(* Logix 5000 project; controller ARS14002_PLC vendor 1 type 14 code 218 rev 30.11; software revision 30.01; part 5 of 13 *)
(* tags used below, declared in another part *)
   AN_1000C : CM_AI_SCL;
   AN_1000C_RESTART_TMR : TIMER;
   AN_1000C_SP : INT;
   AN_1000C_STOP_TMR : TIMER;
   AN_101_PERMISSIVE_AUTO : BOOL;   // Does the PLC look at AN-101
   AN_101A : CM_AI_SCL;
   AN_101A_RESTART_TIME : REAL;
   AN_101A_RESTART_TMR : TIMER;
   AN_101A_SP : REAL;
   AN_101A_STOP_TIME : REAL;
   AN_101A_STOP_TMR : TIMER;
   AN_101B : CM_AI_SCL;
   AN_101B_RESTART_TIME : REAL;
   AN_101B_RESTART_TMR : TIMER;
   AN_101B_SP : REAL;
   AN_101B_STOP_TIME : REAL;
   AN_101B_STOP_TMR : TIMER;
   AN_101C : CM_AI_SCL;
   AN_101C_RESTART_TIME : REAL;
   AN_101C_RESTART_TMR : TIMER;
   AN_101C_SP : REAL;
   AN_101C_STOP_TIME : REAL;
   AN_101C_STOP_TMR : TIMER;
   AN_200A : CM_AI_SCL;
   AN_200A_RESTART_TMR : TIMER;
   AN_200A_SP : REAL;
   AN_200A_STOP_TMR : TIMER;
   ARS_COLLECT : BOOL;
   ARS_COLLECT_AUTO : BOOL;
   ARS_DERIME_AUTO : BOOL;
   AT2_ATOMIZE_LATCH : BOOL;
   AT2_CHAMBER_PRESSURE : REAL;
   AT2_CHAMBER_PRESSURE_SP : REAL;
   AT2_PLANT_ATOMIZING : BOOL;
   AT2_PLANT_BACKFILL : BOOL;
   AT2_PLANT_COLLECT_AUTO : BOOL;
   AT2_PT_101B_Pressure_Override : REAL;   // Setpoint at which FCV_101 will open and relieve the pressure despite controls, not an interlock
   AT2_START_ATOMIZATION : BOOL;
   AT2_V1_OPEN : BOOL;
   AT2_V1_OPEN_POSTHEAT_CTR : COUNTER;
   AT2_V1_OPEN_POSTHEAT_CTR_SP : DINT;
   AT3_ATOMIZE_VALVE_OPEN : BOOL;
   AT3_CHAMBER_PRESSURE : REAL;
   AT3_CHAMBER_PRESSURE_SP : REAL;
   AT3_PLANT_ATOMIZING : BOOL;
   AT3_PLANT_BACKFILL : BOOL;
   AT3_PLANT_COLLECT_AUTO : BOOL;
   AT3_PT_101C_Press_Override : REAL;   // Pressure at which FCV101 will open despite the control scheme, not an interlock
   AT3_V1_OPEN : BOOL;
   Collect_Stop_AT2_O2 : BOOL;
   Collect_Stop_AT3_O2 : BOOL;
   Collect_Stop_Dew_Pt : BOOL;
   COLLECT_STOP_INIT : TIMER;
   Collect_Stop_O2 : BOOL;
   Collect_Stop_PILOT_O2 : BOOL;
   FCV_101A : CM_AO_VLV;
   FCV_101A_DLA : REAL;
   FCV_101A_DLA_BUMP_TMR : TIMER;
   FCV_101A_DLA_TMR : TIMER;
   FCV_101A_STARTPOS : REAL;
   FCV_101B : CM_AO_VLV;
   FCV_101B_DLA : REAL;
   FCV_101B_DLA_BUMP_TMR : TIMER;
   FCV_101B_DLA_TMR : TIMER;
   FCV_101B_STARTPOS : REAL;
   FCV_101C : CM_AO_VLV;
   FCV_101C_DLA : REAL;
   FCV_101C_DLA_BUMP_TMR : TIMER;
   FCV_101C_DLA_TMR : TIMER;
   FCV_101C_STARTPOS : REAL;
   FCV_102A : CM_AO_VLV;
   FCV_102A_AT_STARTPOS : BOOL;
   FCV_102A_SP_Atomize_Venting : REAL;
   FCV_102A_SP_Idle_Collecting : REAL;
   FCV_102A_STARTPOS : REAL;
   FCV_102A_STARTPOS_TIMEOUT : TIMER;
   FCV_102B : CM_AO_VLV;
   FCV_102B_AT_STARTPOS : BOOL;
   FCV_102B_SP_Atomize_Venting : REAL;
   FCV_102B_SP_Idle_Collecting : REAL;
   FCV_102B_STARTPOS : REAL;
   FCV_102B_STARTPOS_TIMEOUT : TIMER;
   FCV_102C : CM_AO_VLV;
   FCV_102C_AT_STARTPOS : BOOL;
   FCV_102C_BUMP_CLOSE_POS : REAL;
   FCV_102C_BUMPED_CLOSED : BOOL;
   FCV_102C_CLOSE_BUMP_TMR : TIMER;
   FCV_102C_SP_Atomize_Venting : REAL;
   FCV_102C_SP_Idle_Collecting : REAL;
   FCV_102C_STARTPOS : REAL;
   FCV_102C_STARTPOS_TIMEOUT : TIMER;
   FCV_204 : CM_AO_VLV;
   FCV_204_AT_STARTPOS : BOOL;
   FCV_204_ATOMIZE_INIT : TIMER;
   FCV_204_PVSWITCH : BOOL;   // 0 = PIT-201 1 = PIT-101C
   FCV_204_SP_Atomize : REAL;
   FCV_204_SP_Atomize_Venting_Only : REAL;
   FCV_204_SP_Idle : REAL;
   FCV_204_STARTPOS : REAL;
   FCV_204_STARTPOS_0 : REAL;
   FCV_STARTPOS_TIMEOUT : TIMER;
   MODE_ATOMIZE : BOOL;
   MODE_IDLE : BOOL;
   MODE_STANDBY_IDLE : BOOL;
   MODE_STANDBY_PUMPUP : BOOL;
   PIDE_101A : PID_ENHANCED;
   PIDE_101B : PID_ENHANCED;
   PIDE_101C : PID_ENHANCED;
   PIDE_102A : PID_ENHANCED;
   PIDE_102B : PID_ENHANCED;
   PIDE_102C : PID_ENHANCED;
   PIDE_204 : PID_ENHANCED;
   PILOT_ATOMIZE_VALVE_OPEN : BOOL;   // Halo Valve
   Pilot_Atomizing_Valve_Close_TON : TIMER;
   Pilot_Atomizing_Valve_Open_TON : TIMER;
   PILOT_EXHAUST_VALVE_OPEN : BOOL;
   PILOT_INLET_VALVE_OPEN : BOOL;   // Pressure Control Status (Backfill)
   Pilot_Inlet_Valve_Open_TON : TIMER;
   PILOT_PLANT_ATOMIZING : BOOL;
   PILOT_PLANT_BACKFILL : BOOL;
   PILOT_PLANT_COLLECT_AUTO : BOOL;
   PILOT_PT_101A_Pressure_Override : REAL;   // Pressure at which 101A will be allowed despite any control limitations, intended as a rescue setpoint, not an interlock
   PT_101A : CM_AI_SCL;
   PT_101B : CM_AI_SCL;
   PT_101C : CM_AI_SCL;
   PT_201 : CM_AI_SCL;
   SV_101AF : CM_DO_GENERIC;
   SV_101AN : CM_DO_GENERIC;
   SV_101AP : CM_DO_GENERIC;
   SV_101BF : CM_DO_GENERIC;
   SV_101BN : CM_DO_GENERIC;
   SV_101BP : CM_DO_GENERIC;
   SV_101CF : CM_DO_GENERIC;
   SV_101CN : CM_DO_GENERIC;
   SV_101CP : CM_DO_GENERIC;
   SV_102AF : CM_DO_GENERIC;
   SV_102BF : CM_DO_GENERIC;
   SV_102CF : CM_DO_GENERIC;
   SV_202F : CM_DO_GENERIC;
   SV_204F : CM_DO_GENERIC;
   TE_501 : CM_AI_SCL;
   TE_501_MIN_SV_202 : REAL;
   TK_700_OVERFULL_DLA_TMR : TIMER;
   XV_101B : CM_DO_VLV;
   XV_101C : CM_DO_VLV;
(* MainProgram, continued *)

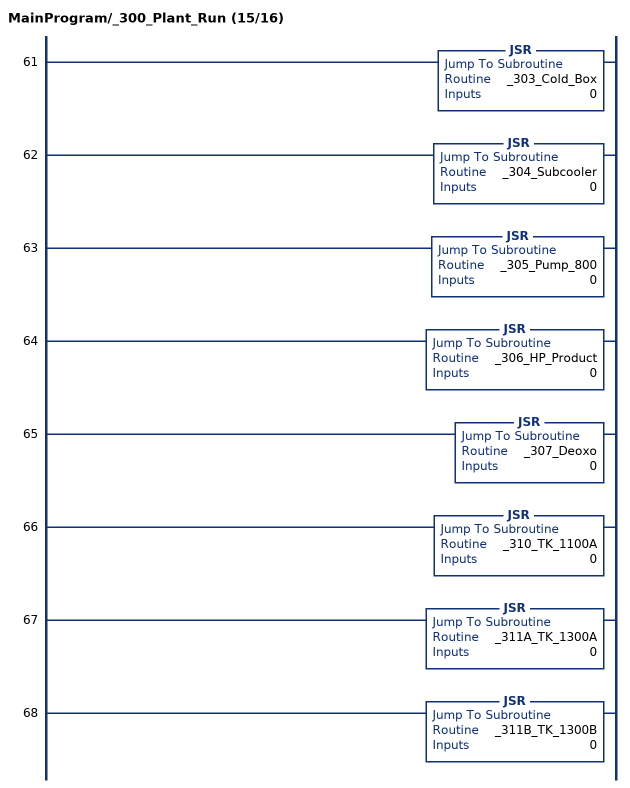
   [picture p83: MainProgram/_300_Plant_Run rungs 61-68]
   61: JSR(_303_Cold_Box,0);
   62: JSR(_304_Subcooler,0);
   63: JSR(_305_Pump_800,0);
   64: JSR(_306_HP_Product,0);
   65: JSR(_307_Deoxo,0);
   66: JSR(_310_TK_1100A,0);
   67: JSR(_311A_TK_1300A,0);
   68: JSR(_311B_TK_1300B,0);
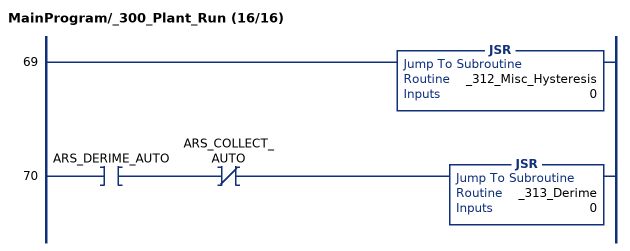
   69: JSR(_312_Misc_Hysteresis,0);
   70: XIC(ARS_DERIME_AUTO)XIO(ARS_COLLECT_AUTO)JSR(_313_Derime,0);
END_ROUTINE

ROUTINE _302_Front_End   (* ladder *)
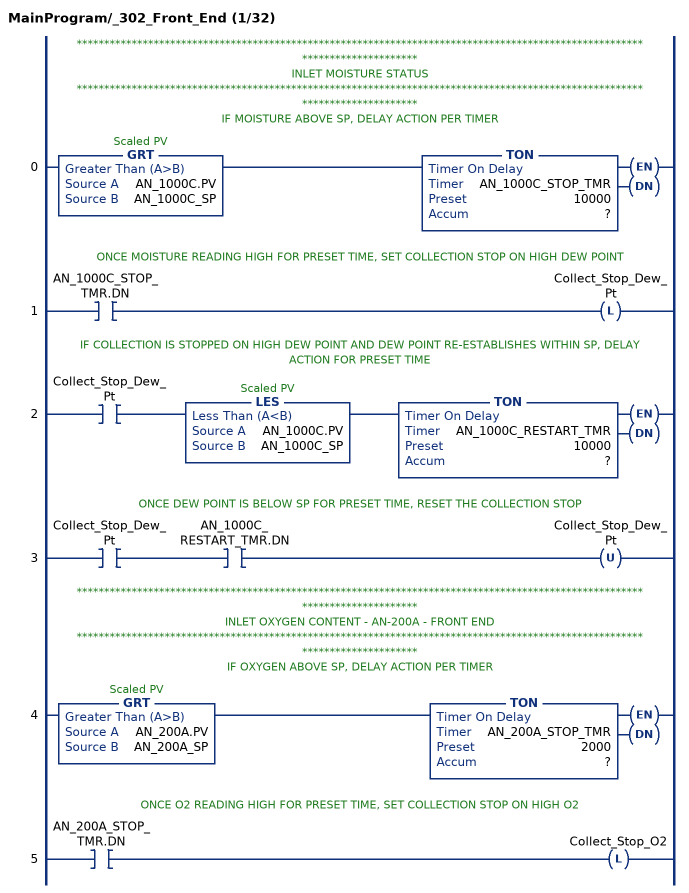
   // ****************************************************************************************************************************
   // INLET MOISTURE STATUS
   // ****************************************************************************************************************************
   // IF MOISTURE ABOVE SP, DELAY ACTION PER TIMER
   0: GRT(AN_1000C.PV,AN_1000C_SP)TON(AN_1000C_STOP_TMR,?,?);
   // ONCE MOISTURE READING HIGH FOR PRESET TIME, SET COLLECTION STOP ON HIGH DEW POINT
   1: XIC(AN_1000C_STOP_TMR.DN)OTL(Collect_Stop_Dew_Pt);
   // IF COLLECTION IS STOPPED ON HIGH DEW POINT AND DEW POINT RE-ESTABLISHES WITHIN SP, DELAY ACTION FOR PRESET TIME
   2: XIC(Collect_Stop_Dew_Pt)LES(AN_1000C.PV,AN_1000C_SP)TON(AN_1000C_RESTART_TMR,?,?);
   // ONCE DEW POINT IS BELOW SP FOR PRESET TIME, RESET THE COLLECTION STOP
   3: XIC(Collect_Stop_Dew_Pt)XIC(AN_1000C_RESTART_TMR.DN)OTU(Collect_Stop_Dew_Pt);
   // ****************************************************************************************************************************
   // INLET OXYGEN CONTENT - AN-200A - FRONT END
   // ****************************************************************************************************************************
   // IF OXYGEN ABOVE SP, DELAY ACTION PER TIMER
   4: GRT(AN_200A.PV,AN_200A_SP)TON(AN_200A_STOP_TMR,?,?);
   // ONCE O2 READING HIGH FOR PRESET TIME, SET COLLECTION STOP ON HIGH O2
   5: XIC(AN_200A_STOP_TMR.DN)OTL(Collect_Stop_O2);
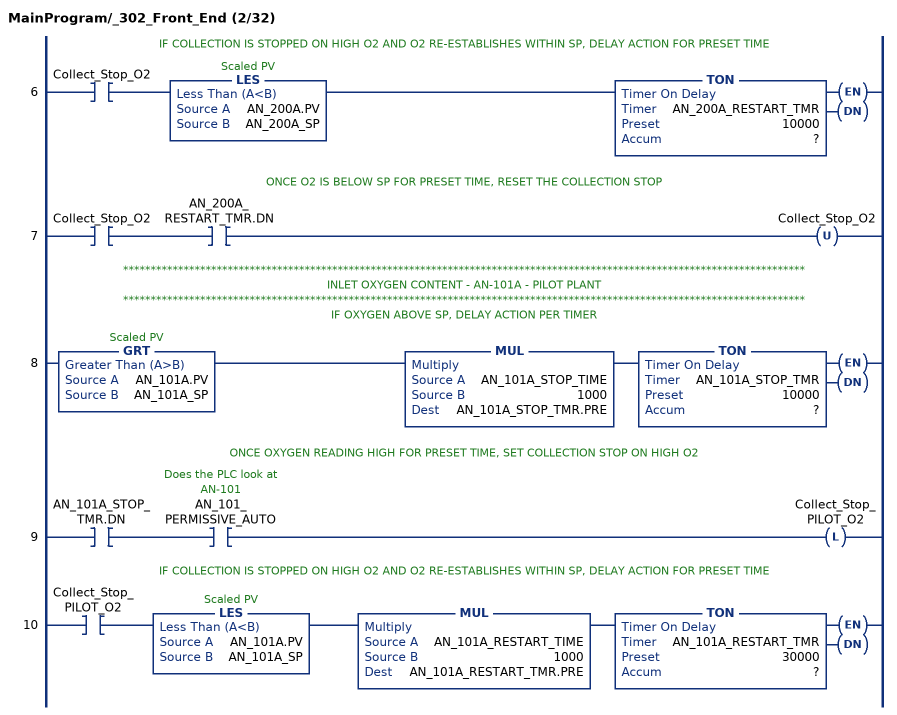
   // IF COLLECTION IS STOPPED ON HIGH O2 AND O2 RE-ESTABLISHES WITHIN SP, DELAY ACTION FOR PRESET TIME
   6: XIC(Collect_Stop_O2)LES(AN_200A.PV,AN_200A_SP)TON(AN_200A_RESTART_TMR,?,?);
   // ONCE O2 IS BELOW SP FOR PRESET TIME, RESET THE COLLECTION STOP
   7: XIC(Collect_Stop_O2)XIC(AN_200A_RESTART_TMR.DN)OTU(Collect_Stop_O2);
   // ****************************************************************************************************************************
   // INLET OXYGEN CONTENT - AN-101A - PILOT PLANT
   // ****************************************************************************************************************************
   // IF OXYGEN ABOVE SP, DELAY ACTION PER TIMER
   8: GRT(AN_101A.PV,AN_101A_SP)MUL(AN_101A_STOP_TIME,1000,AN_101A_STOP_TMR.PRE)TON(AN_101A_STOP_TMR,?,?);
   // ONCE OXYGEN READING HIGH FOR PRESET TIME, SET COLLECTION STOP ON HIGH O2
   9: XIC(AN_101A_STOP_TMR.DN)XIC(AN_101_PERMISSIVE_AUTO)OTL(Collect_Stop_PILOT_O2);
   // IF COLLECTION IS STOPPED ON HIGH O2 AND O2 RE-ESTABLISHES WITHIN SP, DELAY ACTION FOR PRESET TIME
   10: XIC(Collect_Stop_PILOT_O2)LES(AN_101A.PV,AN_101A_SP)MUL(AN_101A_RESTART_TIME,1000,AN_101A_RESTART_TMR.PRE)TON(AN_101A_RESTART_TMR,?,?);
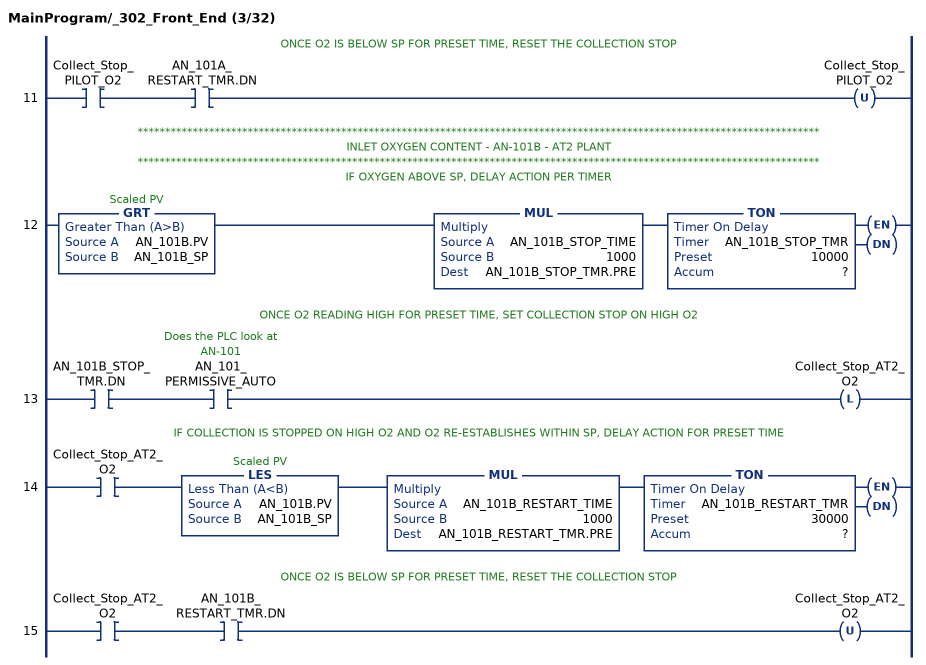
   // ONCE O2 IS BELOW SP FOR PRESET TIME, RESET THE COLLECTION STOP
   11: XIC(Collect_Stop_PILOT_O2)XIC(AN_101A_RESTART_TMR.DN)OTU(Collect_Stop_PILOT_O2);
   // ****************************************************************************************************************************
   // INLET OXYGEN CONTENT - AN-101B - AT2 PLANT
   // ****************************************************************************************************************************
   // IF OXYGEN ABOVE SP, DELAY ACTION PER TIMER
   12: GRT(AN_101B.PV,AN_101B_SP)MUL(AN_101B_STOP_TIME,1000,AN_101B_STOP_TMR.PRE)TON(AN_101B_STOP_TMR,?,?);
   // ONCE O2 READING HIGH FOR PRESET TIME, SET COLLECTION STOP ON HIGH O2
   13: XIC(AN_101B_STOP_TMR.DN)XIC(AN_101_PERMISSIVE_AUTO)OTL(Collect_Stop_AT2_O2);
   // IF COLLECTION IS STOPPED ON HIGH O2 AND O2 RE-ESTABLISHES WITHIN SP, DELAY ACTION FOR PRESET TIME
   14: XIC(Collect_Stop_AT2_O2)LES(AN_101B.PV,AN_101B_SP)MUL(AN_101B_RESTART_TIME,1000,AN_101B_RESTART_TMR.PRE)TON(AN_101B_RESTART_TMR,?,?);
   // ONCE O2 IS BELOW SP FOR PRESET TIME, RESET THE COLLECTION STOP
   15: XIC(Collect_Stop_AT2_O2)XIC(AN_101B_RESTART_TMR.DN)OTU(Collect_Stop_AT2_O2);
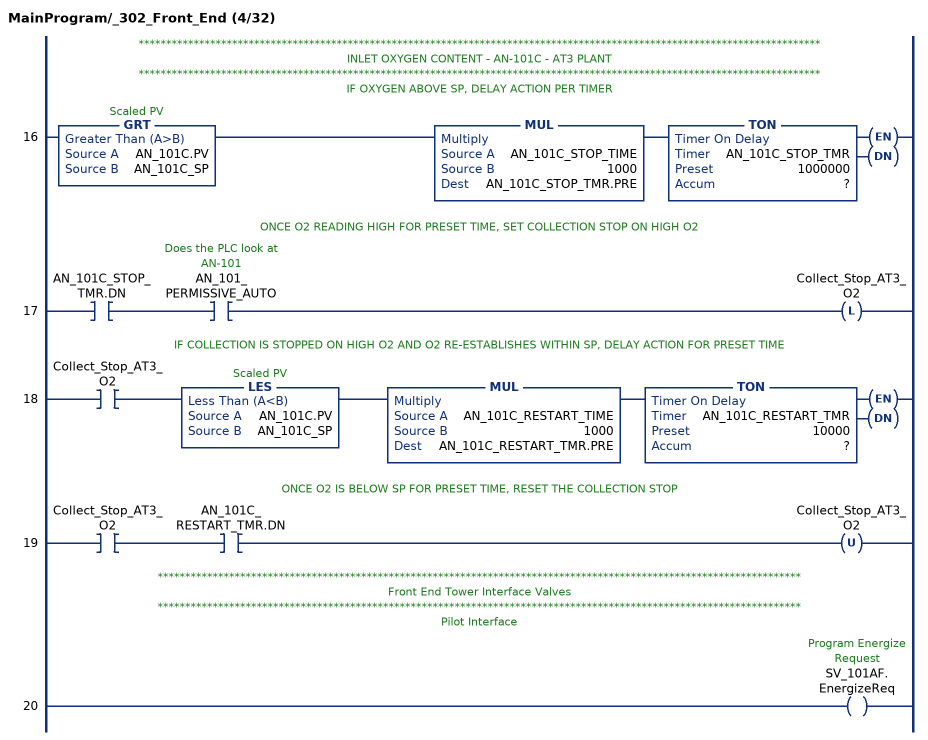
   // ****************************************************************************************************************************
   // INLET OXYGEN CONTENT - AN-101C - AT3 PLANT
   // ****************************************************************************************************************************
   // IF OXYGEN ABOVE SP, DELAY ACTION PER TIMER
   16: GRT(AN_101C.PV,AN_101C_SP)MUL(AN_101C_STOP_TIME,1000,AN_101C_STOP_TMR.PRE)TON(AN_101C_STOP_TMR,?,?);
   // ONCE O2 READING HIGH FOR PRESET TIME, SET COLLECTION STOP ON HIGH O2
   17: XIC(AN_101C_STOP_TMR.DN)XIC(AN_101_PERMISSIVE_AUTO)OTL(Collect_Stop_AT3_O2);
   // IF COLLECTION IS STOPPED ON HIGH O2 AND O2 RE-ESTABLISHES WITHIN SP, DELAY ACTION FOR PRESET TIME
   18: XIC(Collect_Stop_AT3_O2)LES(AN_101C.PV,AN_101C_SP)MUL(AN_101C_RESTART_TIME,1000,AN_101C_RESTART_TMR.PRE)TON(AN_101C_RESTART_TMR,?,?);
   // ONCE O2 IS BELOW SP FOR PRESET TIME, RESET THE COLLECTION STOP
   19: XIC(Collect_Stop_AT3_O2)XIC(AN_101C_RESTART_TMR.DN)OTU(Collect_Stop_AT3_O2);
   // *********************************************************************************************************************
   // Front End Tower Interface Valves
   // *********************************************************************************************************************
   // Pilot Interface
   20: OTE(SV_101AF.EnergizeReq);
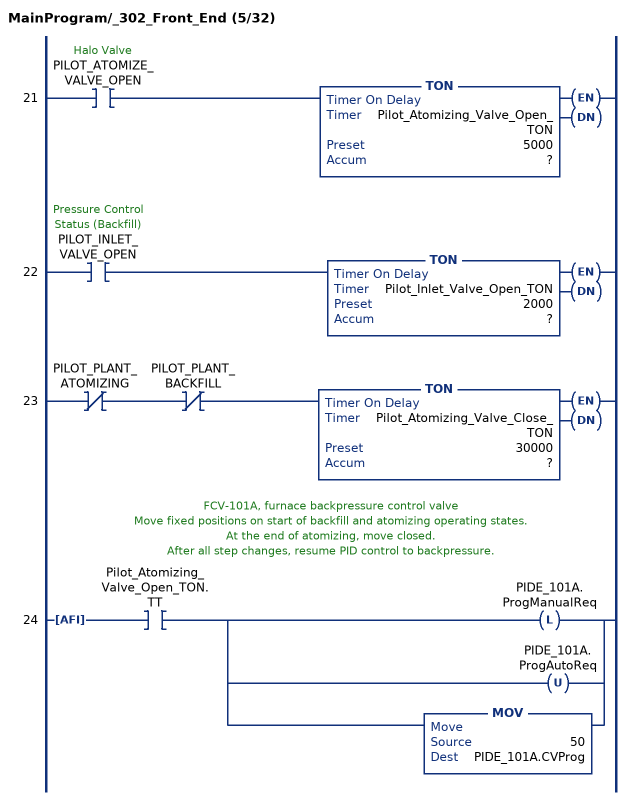
   21: XIC(PILOT_ATOMIZE_VALVE_OPEN)TON(Pilot_Atomizing_Valve_Open_TON,?,?);
   22: XIC(PILOT_INLET_VALVE_OPEN)TON(Pilot_Inlet_Valve_Open_TON,?,?);
   23: XIO(PILOT_PLANT_ATOMIZING)XIO(PILOT_PLANT_BACKFILL)TON(Pilot_Atomizing_Valve_Close_TON,?,?);
   // FCV-101A, furnace backpressure control valve
   // Move fixed positions on start of backfill and atomizing operating states.
   // At the end of atomizing, move closed.
   // After all step changes, resume PID control to backpressure.
   24: AFI()XIC(Pilot_Atomizing_Valve_Open_TON.TT)[OTL(PIDE_101A.ProgManualReq) ,OTU(PIDE_101A.ProgAutoReq) ,MOV(50,PIDE_101A.CVProg) ];
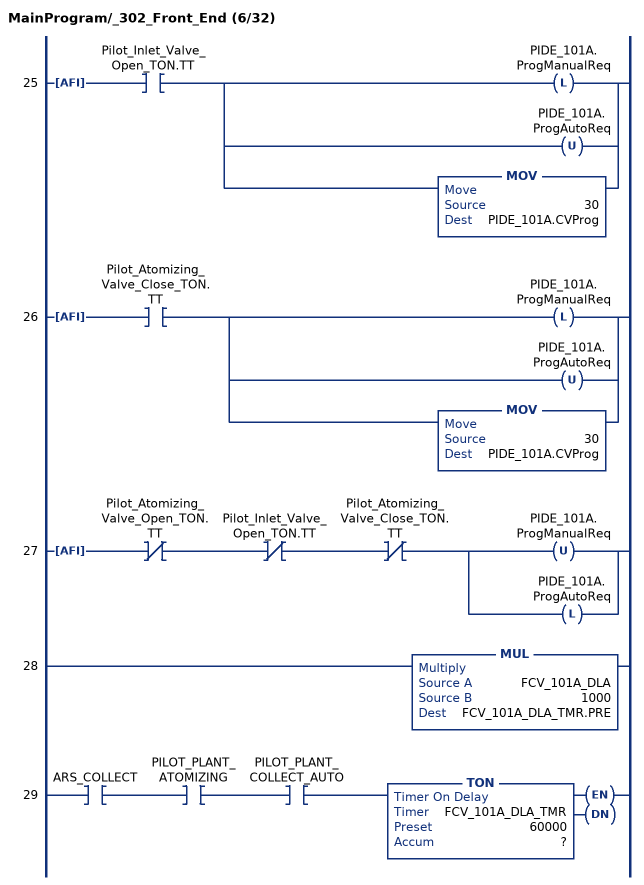
   25: AFI()XIC(Pilot_Inlet_Valve_Open_TON.TT)[OTL(PIDE_101A.ProgManualReq) ,OTU(PIDE_101A.ProgAutoReq) ,MOV(30,PIDE_101A.CVProg) ];
   26: AFI()XIC(Pilot_Atomizing_Valve_Close_TON.TT)[OTL(PIDE_101A.ProgManualReq) ,OTU(PIDE_101A.ProgAutoReq) ,MOV(30,PIDE_101A.CVProg) ];
   27: AFI()XIO(Pilot_Atomizing_Valve_Open_TON.TT)XIO(Pilot_Inlet_Valve_Open_TON.TT)XIO(Pilot_Atomizing_Valve_Close_TON.TT)[OTU(PIDE_101A.ProgManualReq) ,OTL(PIDE_101A.ProgAutoReq) ];
   28: MUL(FCV_101A_DLA,1000,FCV_101A_DLA_TMR.PRE);
   29: XIC(ARS_COLLECT)XIC(PILOT_PLANT_ATOMIZING)XIC(PILOT_PLANT_COLLECT_AUTO)TON(FCV_101A_DLA_TMR,?,?);
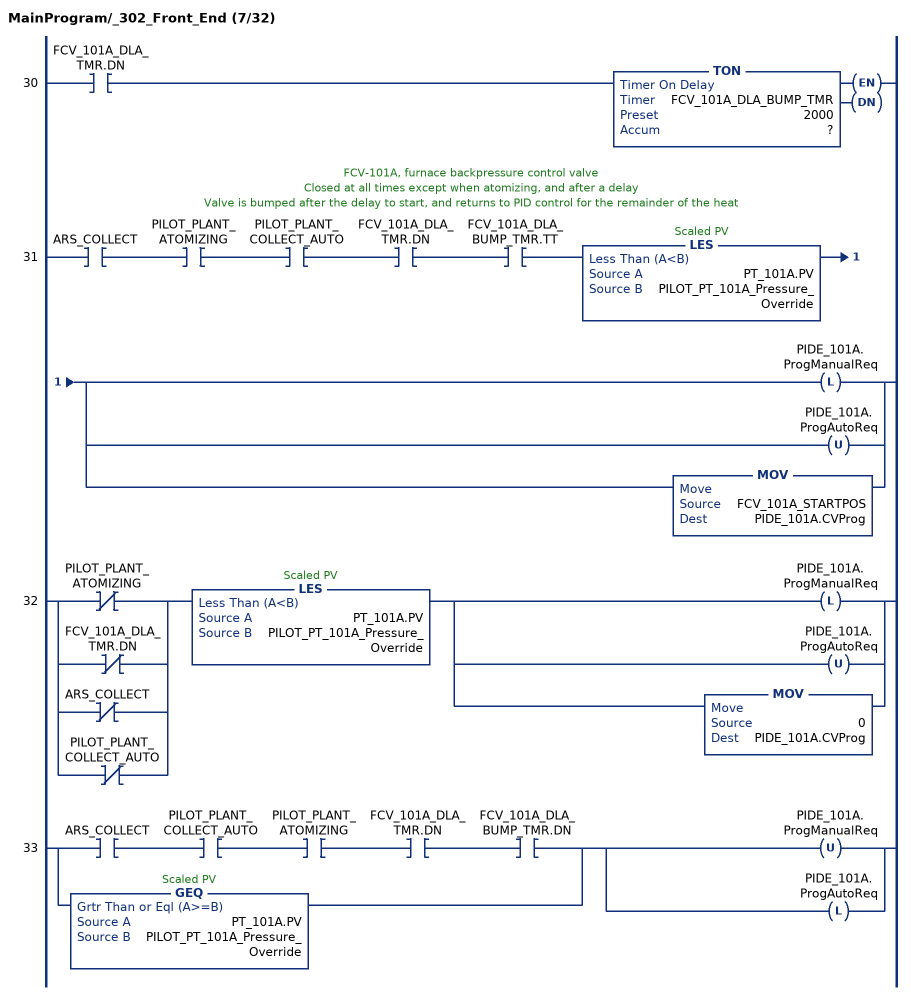
   30: XIC(FCV_101A_DLA_TMR.DN)TON(FCV_101A_DLA_BUMP_TMR,?,?);
   // FCV-101A, furnace backpressure control valve
   // Closed at all times except when atomizing, and after a delay
   // Valve is bumped after the delay to start, and returns to PID control for the remainder of the heat
   31: XIC(ARS_COLLECT)XIC(PILOT_PLANT_ATOMIZING)XIC(PILOT_PLANT_COLLECT_AUTO)XIC(FCV_101A_DLA_TMR.DN)XIC(FCV_101A_DLA_BUMP_TMR.TT)LES(PT_101A.PV,PILOT_PT_101A_Pressure_Override)[OTL(PIDE_101A.ProgManualReq) ,OTU(PIDE_101A.ProgAutoReq) ,MOV(FCV_101A_STARTPOS,PIDE_101A.CVProg) ];
   32: [XIO(PILOT_PLANT_ATOMIZING) ,XIO(FCV_101A_DLA_TMR.DN) ,XIO(ARS_COLLECT) ,XIO(PILOT_PLANT_COLLECT_AUTO) ]LES(PT_101A.PV,PILOT_PT_101A_Pressure_Override)[OTL(PIDE_101A.ProgManualReq) ,OTU(PIDE_101A.ProgAutoReq) ,MOV(0,PIDE_101A.CVProg) ];
   33: [XIC(ARS_COLLECT) XIC(PILOT_PLANT_COLLECT_AUTO) XIC(PILOT_PLANT_ATOMIZING) XIC(FCV_101A_DLA_TMR.DN) XIC(FCV_101A_DLA_BUMP_TMR.DN) ,GEQ(PT_101A.PV,PILOT_PT_101A_Pressure_Override) ][OTU(PIDE_101A.ProgManualReq) ,OTL(PIDE_101A.ProgAutoReq) ];
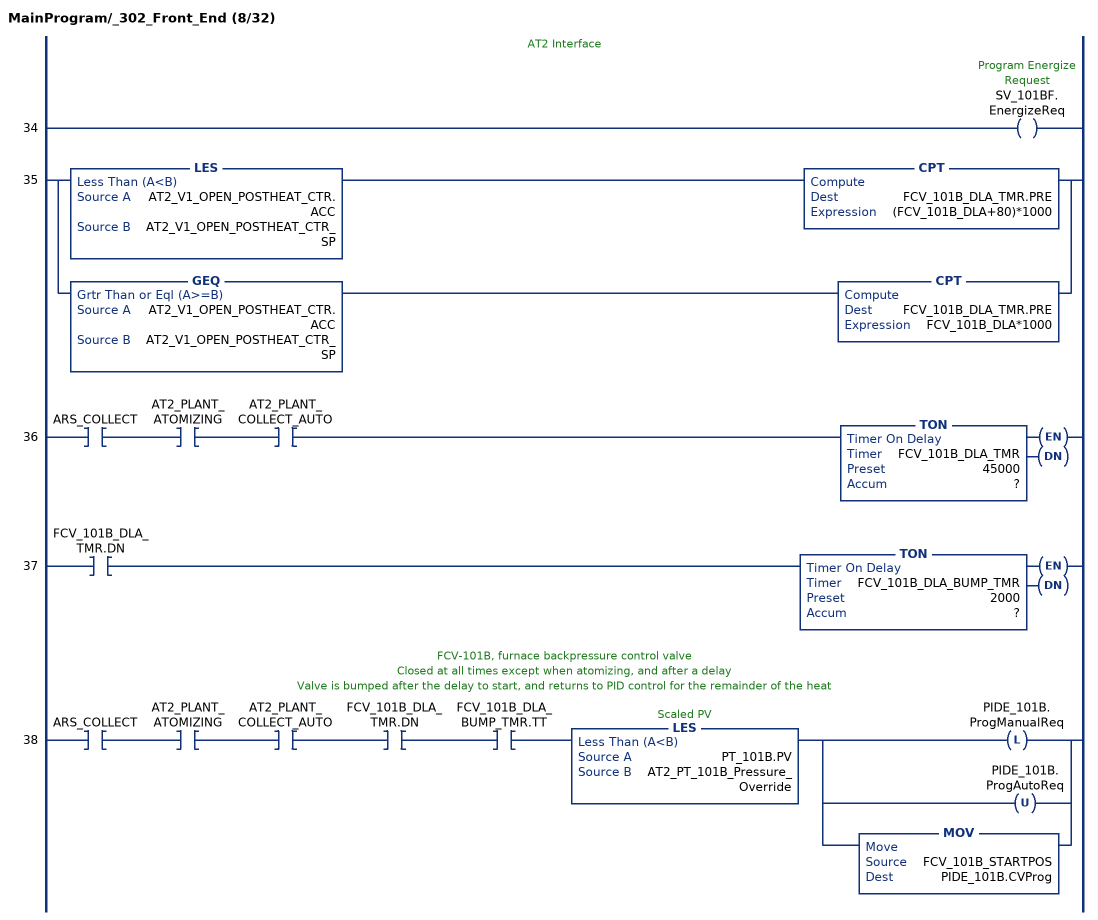
   // AT2 Interface
   34: OTE(SV_101BF.EnergizeReq);
   35: [LES(AT2_V1_OPEN_POSTHEAT_CTR.ACC,AT2_V1_OPEN_POSTHEAT_CTR_SP) CPT(FCV_101B_DLA_TMR.PRE,(FCV_101B_DLA+80)*1000) ,GEQ(AT2_V1_OPEN_POSTHEAT_CTR.ACC,AT2_V1_OPEN_POSTHEAT_CTR_SP) CPT(FCV_101B_DLA_TMR.PRE,FCV_101B_DLA*1000) ];
   36: XIC(ARS_COLLECT)XIC(AT2_PLANT_ATOMIZING)XIC(AT2_PLANT_COLLECT_AUTO)TON(FCV_101B_DLA_TMR,?,?);
   37: XIC(FCV_101B_DLA_TMR.DN)TON(FCV_101B_DLA_BUMP_TMR,?,?);
   // FCV-101B, furnace backpressure control valve
   // Closed at all times except when atomizing, and after a delay
   // Valve is bumped after the delay to start, and returns to PID control for the remainder of the heat
   38: XIC(ARS_COLLECT)XIC(AT2_PLANT_ATOMIZING)XIC(AT2_PLANT_COLLECT_AUTO)XIC(FCV_101B_DLA_TMR.DN)XIC(FCV_101B_DLA_BUMP_TMR.TT)LES(PT_101B.PV,AT2_PT_101B_Pressure_Override)[OTL(PIDE_101B.ProgManualReq) ,OTU(PIDE_101B.ProgAutoReq) ,MOV(FCV_101B_STARTPOS,PIDE_101B.CVProg) ];
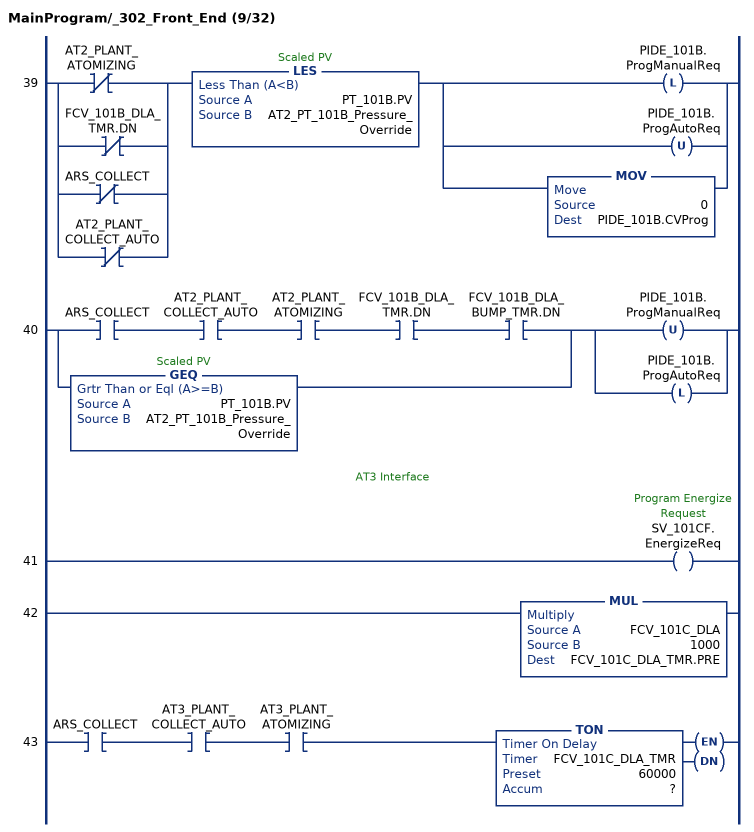
   39: [XIO(AT2_PLANT_ATOMIZING) ,XIO(FCV_101B_DLA_TMR.DN) ,XIO(ARS_COLLECT) ,XIO(AT2_PLANT_COLLECT_AUTO) ]LES(PT_101B.PV,AT2_PT_101B_Pressure_Override)[OTL(PIDE_101B.ProgManualReq) ,OTU(PIDE_101B.ProgAutoReq) ,MOV(0,PIDE_101B.CVProg) ];
   40: [XIC(ARS_COLLECT) XIC(AT2_PLANT_COLLECT_AUTO) XIC(AT2_PLANT_ATOMIZING) XIC(FCV_101B_DLA_TMR.DN) XIC(FCV_101B_DLA_BUMP_TMR.DN) ,GEQ(PT_101B.PV,AT2_PT_101B_Pressure_Override) ][OTU(PIDE_101B.ProgManualReq) ,OTL(PIDE_101B.ProgAutoReq) ];
   // AT3 Interface
   41: OTE(SV_101CF.EnergizeReq);
   42: MUL(FCV_101C_DLA,1000,FCV_101C_DLA_TMR.PRE);
   43: XIC(ARS_COLLECT)XIC(AT3_PLANT_COLLECT_AUTO)XIC(AT3_PLANT_ATOMIZING)TON(FCV_101C_DLA_TMR,?,?);
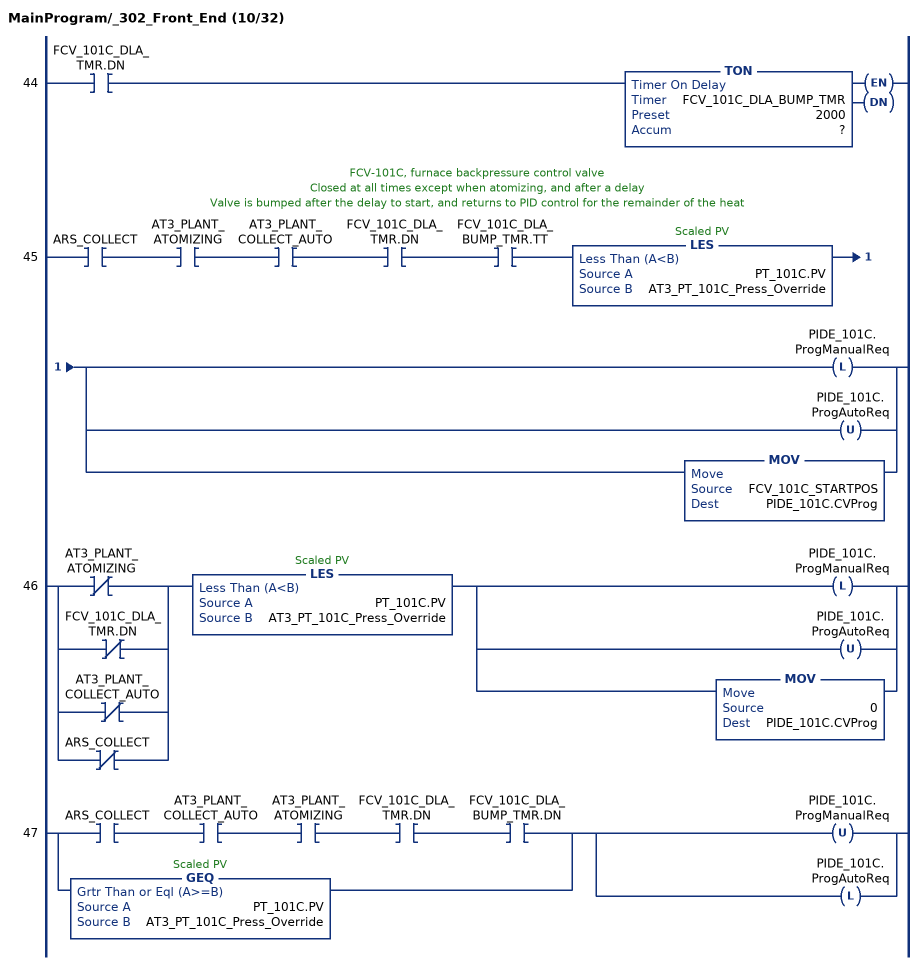
   44: XIC(FCV_101C_DLA_TMR.DN)TON(FCV_101C_DLA_BUMP_TMR,?,?);
   // FCV-101C, furnace backpressure control valve
   // Closed at all times except when atomizing, and after a delay
   // Valve is bumped after the delay to start, and returns to PID control for the remainder of the heat
   45: XIC(ARS_COLLECT)XIC(AT3_PLANT_ATOMIZING)XIC(AT3_PLANT_COLLECT_AUTO)XIC(FCV_101C_DLA_TMR.DN)XIC(FCV_101C_DLA_BUMP_TMR.TT)LES(PT_101C.PV,AT3_PT_101C_Press_Override)[OTL(PIDE_101C.ProgManualReq) ,OTU(PIDE_101C.ProgAutoReq) ,MOV(FCV_101C_STARTPOS,PIDE_101C.CVProg) ];
   46: [XIO(AT3_PLANT_ATOMIZING) ,XIO(FCV_101C_DLA_TMR.DN) ,XIO(AT3_PLANT_COLLECT_AUTO) ,XIO(ARS_COLLECT) ]LES(PT_101C.PV,AT3_PT_101C_Press_Override)[OTL(PIDE_101C.ProgManualReq) ,OTU(PIDE_101C.ProgAutoReq) ,MOV(0,PIDE_101C.CVProg) ];
   47: [XIC(ARS_COLLECT) XIC(AT3_PLANT_COLLECT_AUTO) XIC(AT3_PLANT_ATOMIZING) XIC(FCV_101C_DLA_TMR.DN) XIC(FCV_101C_DLA_BUMP_TMR.DN) ,GEQ(PT_101C.PV,AT3_PT_101C_Press_Override) ][OTU(PIDE_101C.ProgManualReq) ,OTL(PIDE_101C.ProgAutoReq) ];
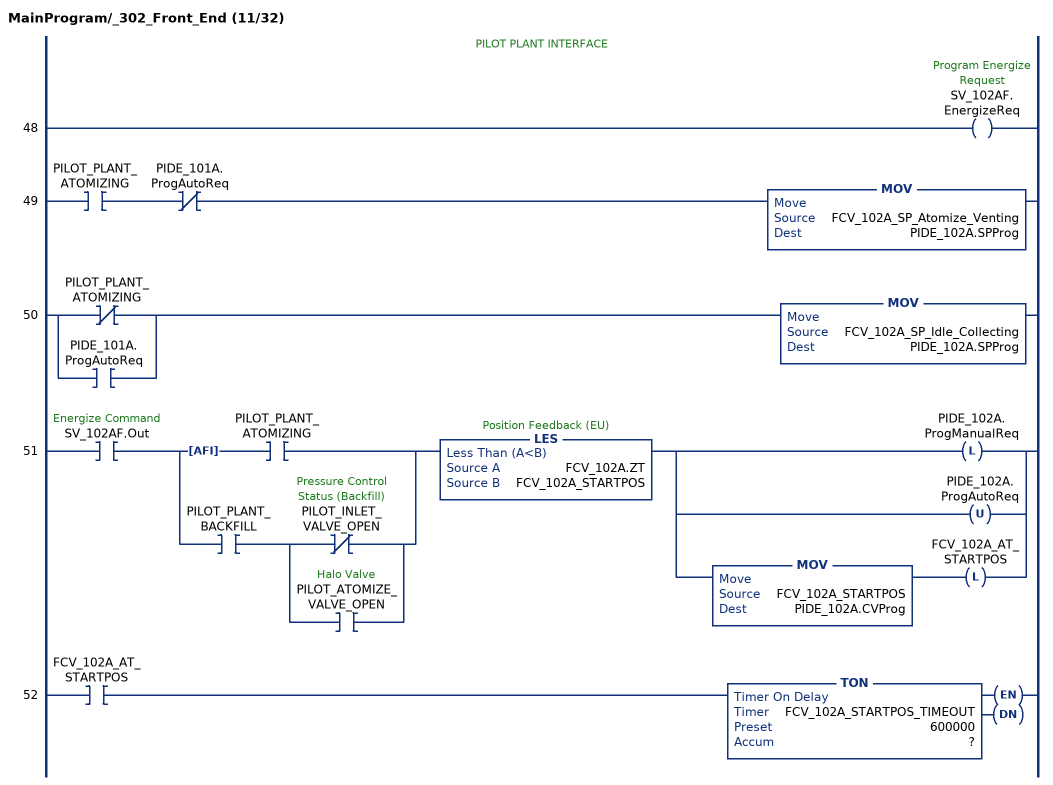
   // PILOT PLANT INTERFACE
   48: OTE(SV_102AF.EnergizeReq);
   49: XIC(PILOT_PLANT_ATOMIZING)XIO(PIDE_101A.ProgAutoReq)MOV(FCV_102A_SP_Atomize_Venting,PIDE_102A.SPProg);
   50: [XIO(PILOT_PLANT_ATOMIZING) ,XIC(PIDE_101A.ProgAutoReq) ]MOV(FCV_102A_SP_Idle_Collecting,PIDE_102A.SPProg);
   51: XIC(SV_102AF.Out)[AFI() XIC(PILOT_PLANT_ATOMIZING) ,XIC(PILOT_PLANT_BACKFILL) [XIO(PILOT_INLET_VALVE_OPEN) ,XIC(PILOT_ATOMIZE_VALVE_OPEN) ] ]LES(FCV_102A.ZT,FCV_102A_STARTPOS)[OTL(PIDE_102A.ProgManualReq) ,OTU(PIDE_102A.ProgAutoReq) ,MOV(FCV_102A_STARTPOS,PIDE_102A.CVProg) OTL(FCV_102A_AT_STARTPOS) ];
   52: XIC(FCV_102A_AT_STARTPOS)TON(FCV_102A_STARTPOS_TIMEOUT,?,?);
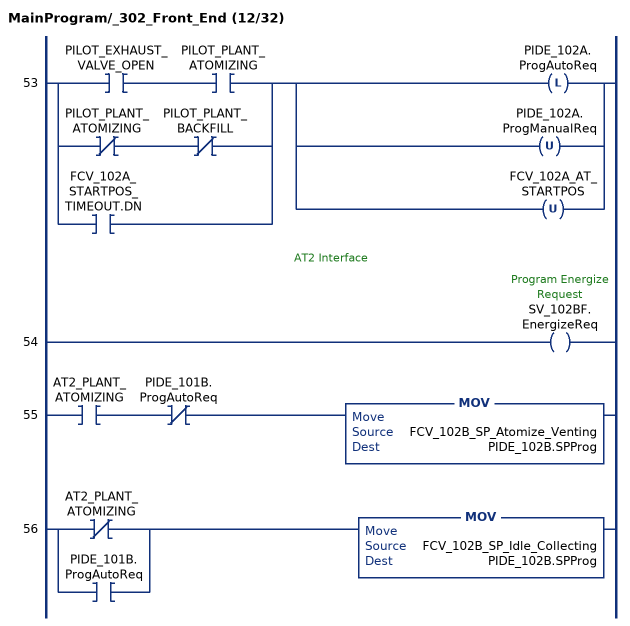
   53: [XIC(PILOT_EXHAUST_VALVE_OPEN) XIC(PILOT_PLANT_ATOMIZING) ,XIO(PILOT_PLANT_ATOMIZING) XIO(PILOT_PLANT_BACKFILL) ,XIC(FCV_102A_STARTPOS_TIMEOUT.DN) ][OTL(PIDE_102A.ProgAutoReq) ,OTU(PIDE_102A.ProgManualReq) ,OTU(FCV_102A_AT_STARTPOS) ];
   // AT2 Interface
   54: OTE(SV_102BF.EnergizeReq);
   55: XIC(AT2_PLANT_ATOMIZING)XIO(PIDE_101B.ProgAutoReq)MOV(FCV_102B_SP_Atomize_Venting,PIDE_102B.SPProg);
   56: [XIO(AT2_PLANT_ATOMIZING) ,XIC(PIDE_101B.ProgAutoReq) ]MOV(FCV_102B_SP_Idle_Collecting,PIDE_102B.SPProg);
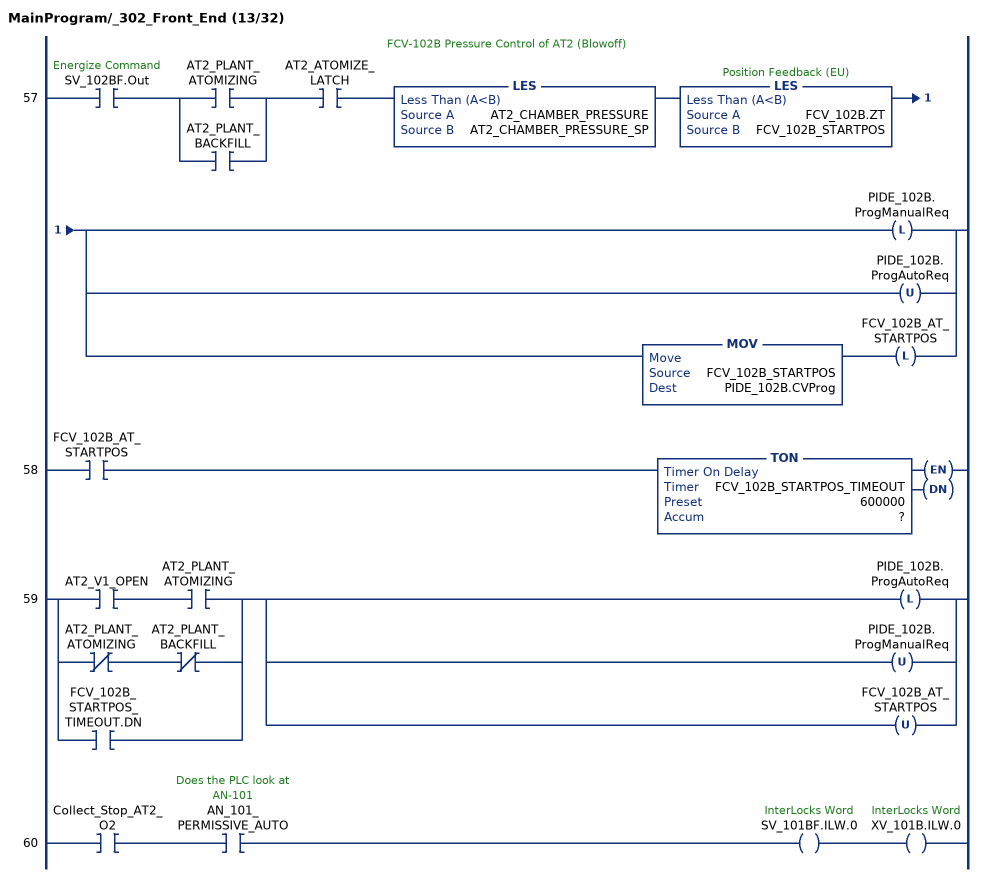
   // FCV-102B Pressure Control of AT2 (Blowoff)
   57: XIC(SV_102BF.Out)[XIC(AT2_PLANT_ATOMIZING) ,XIC(AT2_PLANT_BACKFILL) ]XIC(AT2_ATOMIZE_LATCH)LES(AT2_CHAMBER_PRESSURE,AT2_CHAMBER_PRESSURE_SP)LES(FCV_102B.ZT,FCV_102B_STARTPOS)[OTL(PIDE_102B.ProgManualReq) ,[OTU(PIDE_102B.ProgAutoReq) ,MOV(FCV_102B_STARTPOS,PIDE_102B.CVProg) OTL(FCV_102B_AT_STARTPOS) ] ];
   58: XIC(FCV_102B_AT_STARTPOS)TON(FCV_102B_STARTPOS_TIMEOUT,?,?);
   59: [XIC(AT2_V1_OPEN) XIC(AT2_PLANT_ATOMIZING) ,XIO(AT2_PLANT_ATOMIZING) XIO(AT2_PLANT_BACKFILL) ,XIC(FCV_102B_STARTPOS_TIMEOUT.DN) ][OTL(PIDE_102B.ProgAutoReq) ,OTU(PIDE_102B.ProgManualReq) ,OTU(FCV_102B_AT_STARTPOS) ];
   60: XIC(Collect_Stop_AT2_O2)XIC(AN_101_PERMISSIVE_AUTO)OTE(SV_101BF.ILW.0)OTE(XV_101B.ILW.0);
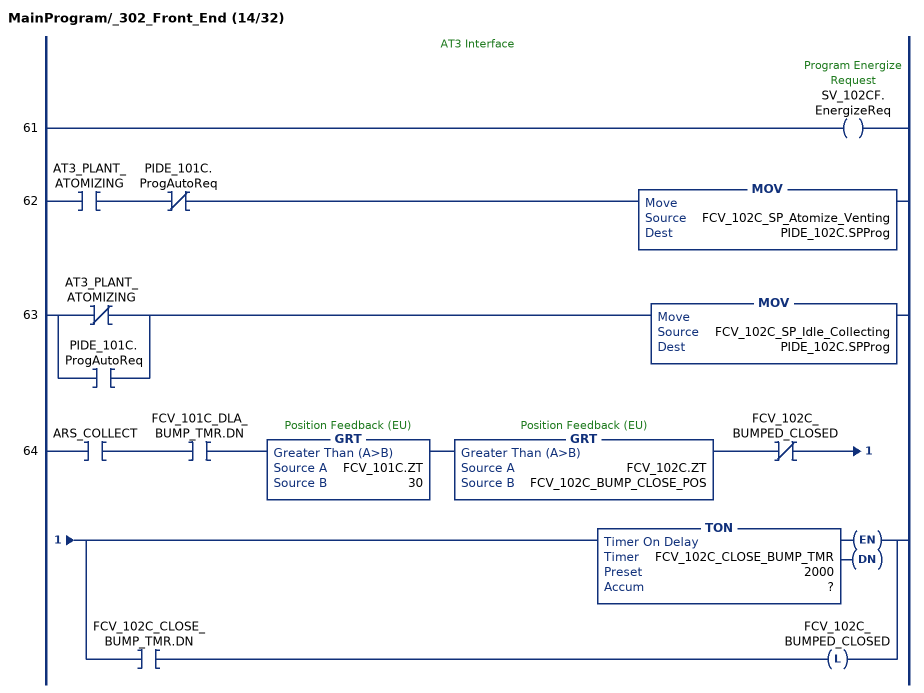
   // AT3 Interface
   61: OTE(SV_102CF.EnergizeReq);
   62: XIC(AT3_PLANT_ATOMIZING)XIO(PIDE_101C.ProgAutoReq)MOV(FCV_102C_SP_Atomize_Venting,PIDE_102C.SPProg);
   63: [XIO(AT3_PLANT_ATOMIZING) ,XIC(PIDE_101C.ProgAutoReq) ]MOV(FCV_102C_SP_Idle_Collecting,PIDE_102C.SPProg);
   64: XIC(ARS_COLLECT)XIC(FCV_101C_DLA_BUMP_TMR.DN)GRT(FCV_101C.ZT,30)GRT(FCV_102C.ZT,FCV_102C_BUMP_CLOSE_POS)XIO(FCV_102C_BUMPED_CLOSED)[TON(FCV_102C_CLOSE_BUMP_TMR,?,?) ,XIC(FCV_102C_CLOSE_BUMP_TMR.DN) OTL(FCV_102C_BUMPED_CLOSED) ];
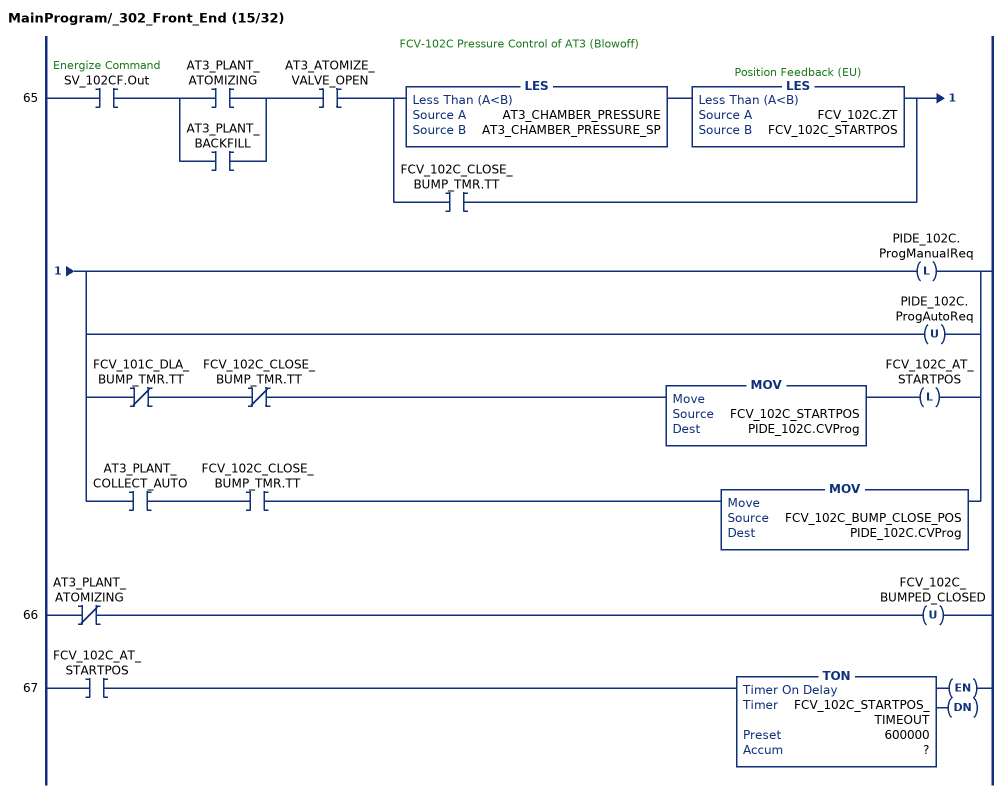
   // FCV-102C Pressure Control of AT3 (Blowoff)
   65: XIC(SV_102CF.Out)[XIC(AT3_PLANT_ATOMIZING) ,XIC(AT3_PLANT_BACKFILL) ]XIC(AT3_ATOMIZE_VALVE_OPEN)[LES(AT3_CHAMBER_PRESSURE,AT3_CHAMBER_PRESSURE_SP) LES(FCV_102C.ZT,FCV_102C_STARTPOS) ,XIC(FCV_102C_CLOSE_BUMP_TMR.TT) ][OTL(PIDE_102C.ProgManualReq) ,[OTU(PIDE_102C.ProgAutoReq) ,XIO(FCV_101C_DLA_BUMP_TMR.TT) XIO(FCV_102C_CLOSE_BUMP_TMR.TT) MOV(FCV_102C_STARTPOS,PIDE_102C.CVProg) OTL(FCV_102C_AT_STARTPOS) ,XIC(AT3_PLANT_COLLECT_AUTO) XIC(FCV_102C_CLOSE_BUMP_TMR.TT) MOV(FCV_102C_BUMP_CLOSE_POS,PIDE_102C.CVProg) ] ];
   66: XIO(AT3_PLANT_ATOMIZING)OTU(FCV_102C_BUMPED_CLOSED);
   67: XIC(FCV_102C_AT_STARTPOS)TON(FCV_102C_STARTPOS_TIMEOUT,?,?);
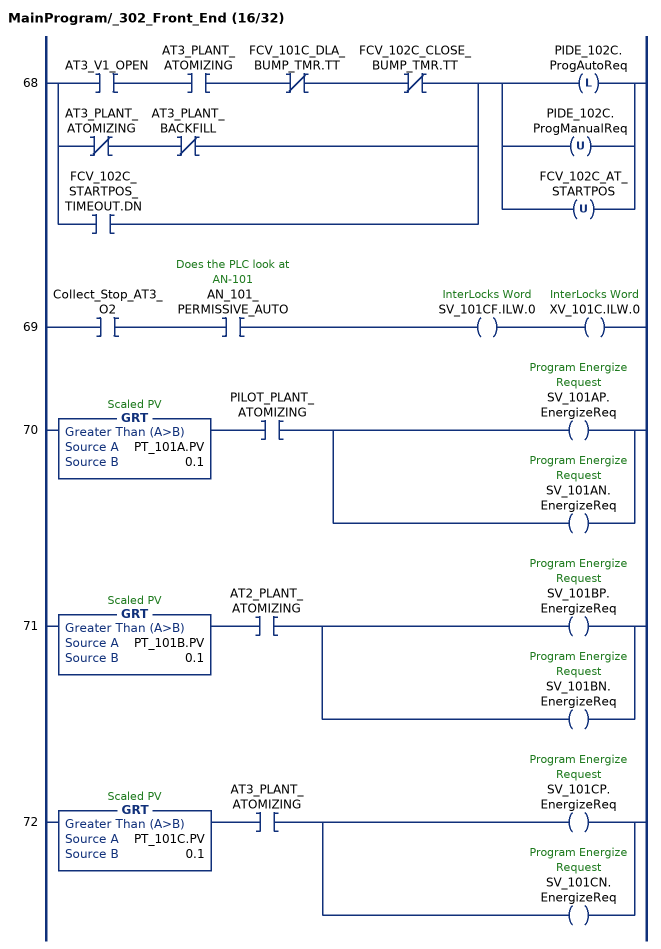
   68: [XIC(AT3_V1_OPEN) XIC(AT3_PLANT_ATOMIZING) XIO(FCV_101C_DLA_BUMP_TMR.TT) XIO(FCV_102C_CLOSE_BUMP_TMR.TT) ,XIO(AT3_PLANT_ATOMIZING) XIO(AT3_PLANT_BACKFILL) ,XIC(FCV_102C_STARTPOS_TIMEOUT.DN) ][OTL(PIDE_102C.ProgAutoReq) ,OTU(PIDE_102C.ProgManualReq) ,OTU(FCV_102C_AT_STARTPOS) ];
   69: XIC(Collect_Stop_AT3_O2)XIC(AN_101_PERMISSIVE_AUTO)OTE(SV_101CF.ILW.0)OTE(XV_101C.ILW.0);
   70: GRT(PT_101A.PV,0.1)XIC(PILOT_PLANT_ATOMIZING)[OTE(SV_101AP.EnergizeReq) ,OTE(SV_101AN.EnergizeReq) ];
   71: GRT(PT_101B.PV,0.1)XIC(AT2_PLANT_ATOMIZING)[OTE(SV_101BP.EnergizeReq) ,OTE(SV_101BN.EnergizeReq) ];
   72: GRT(PT_101C.PV,0.1)XIC(AT3_PLANT_ATOMIZING)[OTE(SV_101CP.EnergizeReq) ,OTE(SV_101CN.EnergizeReq) ];
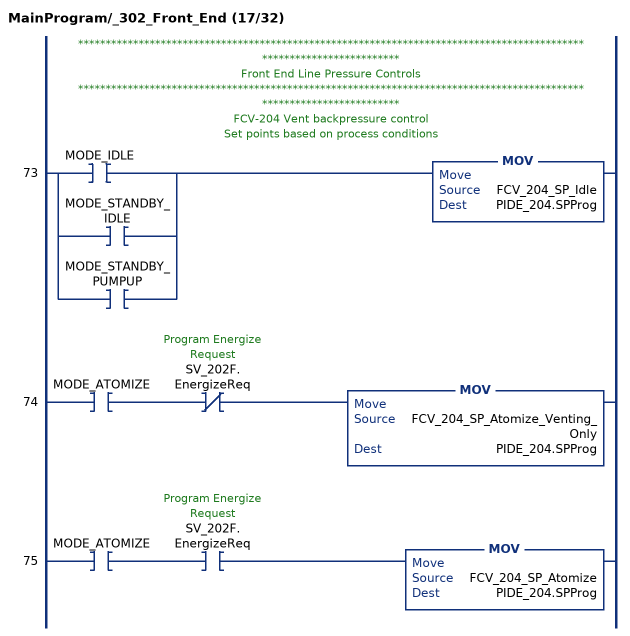
   // *********************************************************************************************************************
   // Front End Line Pressure Controls
   // *********************************************************************************************************************
   // FCV-204 Vent backpressure control
   // Set points based on process conditions
   73: [XIC(MODE_IDLE) ,XIC(MODE_STANDBY_IDLE) ,XIC(MODE_STANDBY_PUMPUP) ]MOV(FCV_204_SP_Idle,PIDE_204.SPProg);
   74: XIC(MODE_ATOMIZE)XIO(SV_202F.EnergizeReq)MOV(FCV_204_SP_Atomize_Venting_Only,PIDE_204.SPProg);
   75: XIC(MODE_ATOMIZE)XIC(SV_202F.EnergizeReq)MOV(FCV_204_SP_Atomize,PIDE_204.SPProg);
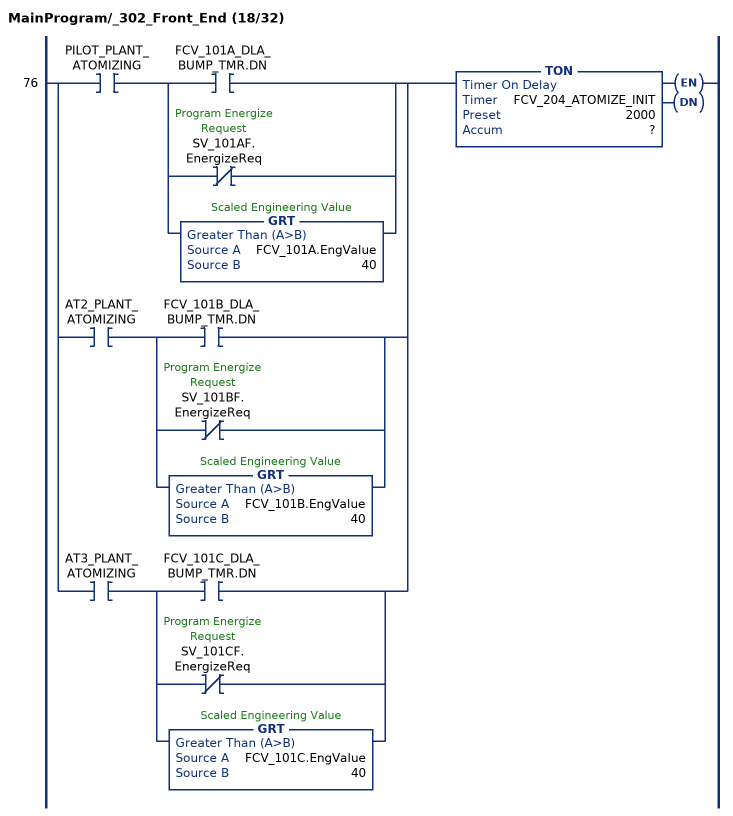
   76: [XIC(PILOT_PLANT_ATOMIZING) [XIC(FCV_101A_DLA_BUMP_TMR.DN) ,XIO(SV_101AF.EnergizeReq) ,GRT(FCV_101A.EngValue,40) ] ,XIC(AT2_PLANT_ATOMIZING) [XIC(FCV_101B_DLA_BUMP_TMR.DN) ,XIO(SV_101BF.EnergizeReq) ,GRT(FCV_101B.EngValue,40) ] ,XIC(AT3_PLANT_ATOMIZING) [XIC(FCV_101C_DLA_BUMP_TMR.DN) ,XIO(SV_101CF.EnergizeReq) ,GRT(FCV_101C.EngValue,40) ] ]TON(FCV_204_ATOMIZE_INIT,?,?);
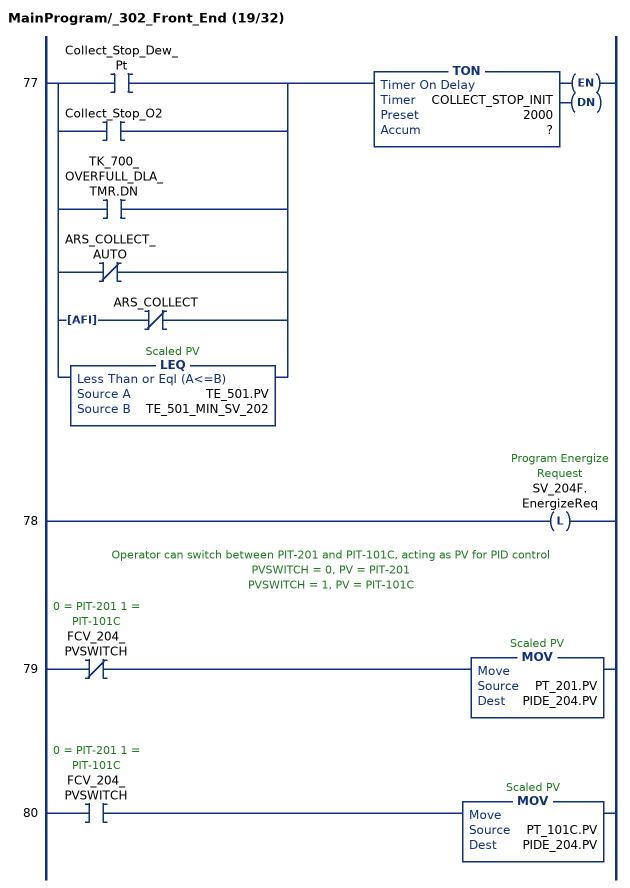
   77: [XIC(Collect_Stop_Dew_Pt) ,XIC(Collect_Stop_O2) ,XIC(TK_700_OVERFULL_DLA_TMR.DN) ,XIO(ARS_COLLECT_AUTO) ,AFI() XIO(ARS_COLLECT) ,LEQ(TE_501.PV,TE_501_MIN_SV_202) ]TON(COLLECT_STOP_INIT,?,?);
   78: OTL(SV_204F.EnergizeReq);
   // Operator can switch between PIT-201 and PIT-101C, acting as PV for PID control
   // PVSWITCH = 0, PV = PIT-201
   // PVSWITCH = 1, PV = PIT-101C
   79: XIO(FCV_204_PVSWITCH)MOV(PT_201.PV,PIDE_204.PV);
   80: XIC(FCV_204_PVSWITCH)MOV(PT_101C.PV,PIDE_204.PV);
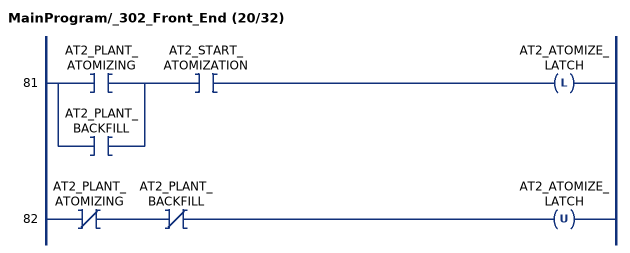
   81: [XIC(AT2_PLANT_ATOMIZING) ,XIC(AT2_PLANT_BACKFILL) ]XIC(AT2_START_ATOMIZATION)OTL(AT2_ATOMIZE_LATCH);
   82: XIO(AT2_PLANT_ATOMIZING)XIO(AT2_PLANT_BACKFILL)OTU(AT2_ATOMIZE_LATCH);
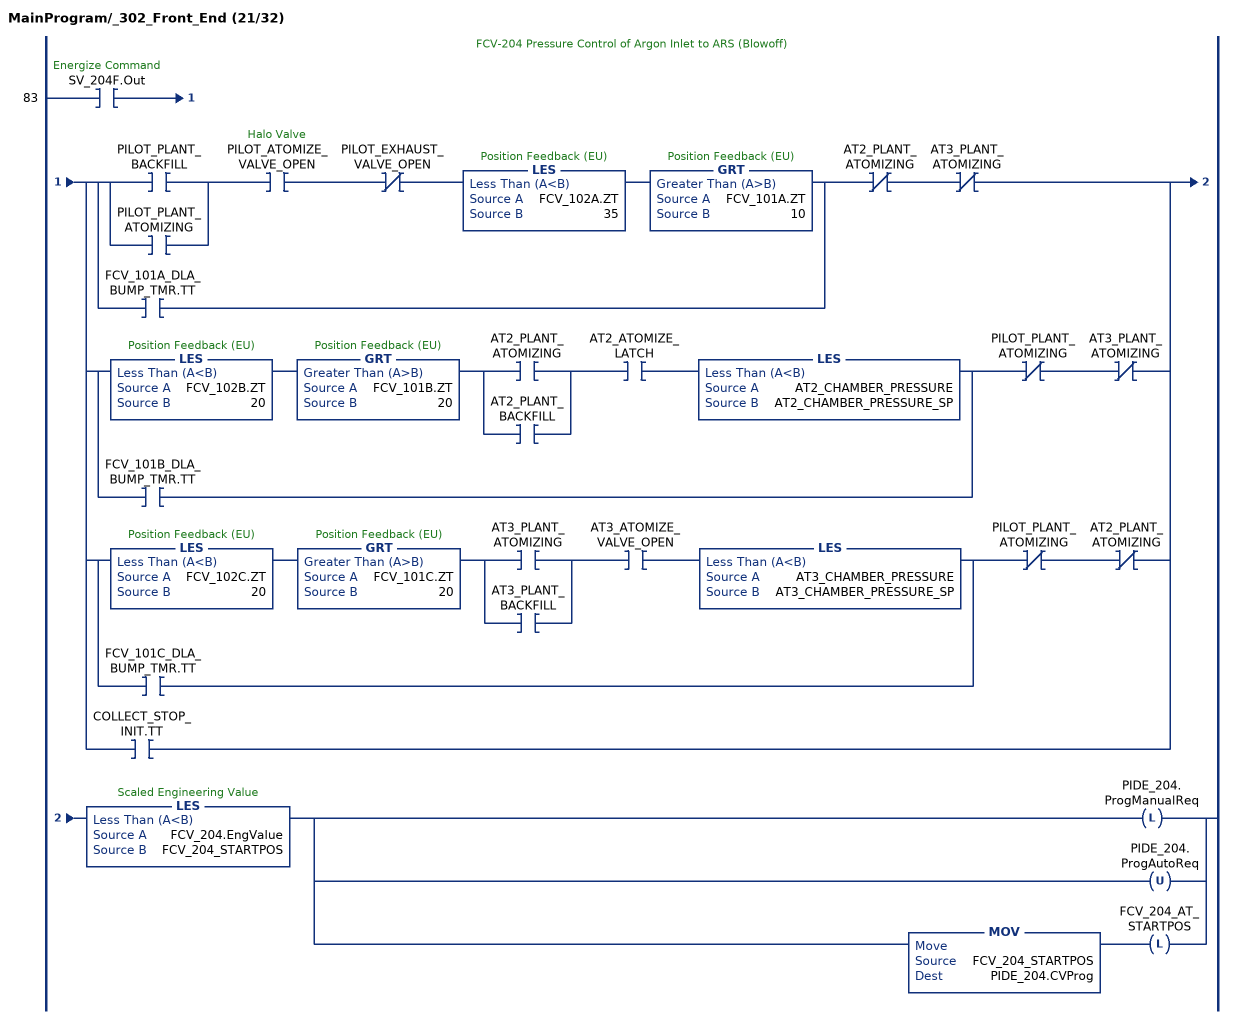
   // FCV-204 Pressure Control of Argon Inlet to ARS (Blowoff)
   83: XIC(SV_204F.Out)[[[XIC(PILOT_PLANT_BACKFILL) ,XIC(PILOT_PLANT_ATOMIZING) ] XIC(PILOT_ATOMIZE_VALVE_OPEN) XIO(PILOT_EXHAUST_VALVE_OPEN) LES(FCV_102A.ZT,35) GRT(FCV_101A.ZT,10) ,XIC(FCV_101A_DLA_BUMP_TMR.TT) ] XIO(AT2_PLANT_ATOMIZING) XIO(AT3_PLANT_ATOMIZING) ,[LES(FCV_102B.ZT,20) GRT(FCV_101B.ZT,20) [XIC(AT2_PLANT_ATOMIZING) ,XIC(AT2_PLANT_BACKFILL) ] XIC(AT2_ATOMIZE_LATCH) LES(AT2_CHAMBER_PRESSURE,AT2_CHAMBER_PRESSURE_SP) ,XIC(FCV_101B_DLA_BUMP_TMR.TT) ] XIO(PILOT_PLANT_ATOMIZING) XIO(AT3_PLANT_ATOMIZING) ,[LES(FCV_102C.ZT,20) GRT(FCV_101C.ZT,20) [XIC(AT3_PLANT_ATOMIZING) ,XIC(AT3_PLANT_BACKFILL) ] XIC(AT3_ATOMIZE_VALVE_OPEN) LES(AT3_CHAMBER_PRESSURE,AT3_CHAMBER_PRESSURE_SP) ,XIC(FCV_101C_DLA_BUMP_TMR.TT) ] XIO(PILOT_PLANT_ATOMIZING) XIO(AT2_PLANT_ATOMIZING) ,XIC(COLLECT_STOP_INIT.TT) ]LES(FCV_204.EngValue,FCV_204_STARTPOS)[OTL(PIDE_204.ProgManualReq) ,[OTU(PIDE_204.ProgAutoReq) ,MOV(FCV_204_STARTPOS,PIDE_204.CVProg) OTL(FCV_204_AT_STARTPOS) ] ];
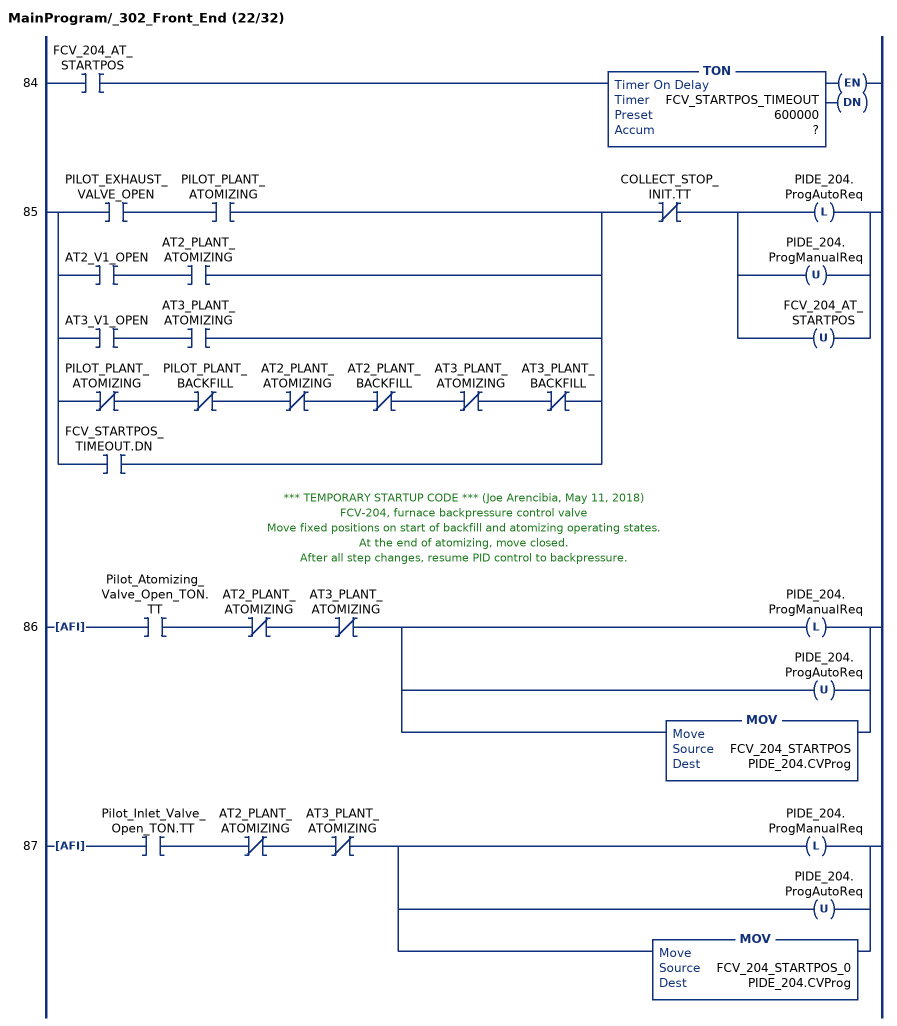
   84: XIC(FCV_204_AT_STARTPOS)TON(FCV_STARTPOS_TIMEOUT,?,?);
   85: [XIC(PILOT_EXHAUST_VALVE_OPEN) XIC(PILOT_PLANT_ATOMIZING) ,XIC(AT2_V1_OPEN) XIC(AT2_PLANT_ATOMIZING) ,XIC(AT3_V1_OPEN) XIC(AT3_PLANT_ATOMIZING) ,XIO(PILOT_PLANT_ATOMIZING) XIO(PILOT_PLANT_BACKFILL) XIO(AT2_PLANT_ATOMIZING) XIO(AT2_PLANT_BACKFILL) XIO(AT3_PLANT_ATOMIZING) XIO(AT3_PLANT_BACKFILL) ,XIC(FCV_STARTPOS_TIMEOUT.DN) ]XIO(COLLECT_STOP_INIT.TT)[OTL(PIDE_204.ProgAutoReq) ,OTU(PIDE_204.ProgManualReq) ,OTU(FCV_204_AT_STARTPOS) ];
   // *** TEMPORARY STARTUP CODE *** (Joe Arencibia, May 11, 2018)
   // FCV-204, furnace backpressure control valve
   // Move fixed positions on start of backfill and atomizing operating states.
   // At the end of atomizing, move closed.
   // After all step changes, resume PID control to backpressure.
   86: AFI()XIC(Pilot_Atomizing_Valve_Open_TON.TT)XIO(AT2_PLANT_ATOMIZING)XIO(AT3_PLANT_ATOMIZING)[OTL(PIDE_204.ProgManualReq) ,OTU(PIDE_204.ProgAutoReq) ,MOV(FCV_204_STARTPOS,PIDE_204.CVProg) ];
   87: AFI()XIC(Pilot_Inlet_Valve_Open_TON.TT)XIO(AT2_PLANT_ATOMIZING)XIO(AT3_PLANT_ATOMIZING)[OTL(PIDE_204.ProgManualReq) ,OTU(PIDE_204.ProgAutoReq) ,MOV(FCV_204_STARTPOS_0,PIDE_204.CVProg) ];
